(* PLC project 117_1_V0.5.project, CODESYS CODESYS V3.5 SP17 Patch 3 *)
(* stored: creationDateTime 1970-01-01T00:00:00, modificationDateTime 2026-03-26T18:14:32.4070562 *)

FUNCTION_BLOCK TimeManager
  VAR
    hTask : CmpIecTask.RTS_IEC_HANDLE;  (* Дескриптор (handle) задачи * ) *)
    result : CmpIecTask.RTS_IEC_RESULT;  (* Результат выполнения функций * ) *)
    pCurrentTaskInfo : POINTER TO CmpIecTask.Task_Info2;  (* Указатель на структуру с информацией о задаче * ) *)
    CurrentTaskInfo : CmpIecTask.Task_Info2;  (* Сама структура с данными * ) *)
    DateAndTime : DTU.GetDateAndTime;
    _dateAndTime : DT;
  END_VAR

            
// 1. Получаем дескриптор текущей задачи
hTask := CmpIecTask.IecTaskGetCurrent(pResult := ADR(result));

// 2. Если дескриптор получен успешно, запрашиваем информацию о задаче
IF hTask <> 0 THEN
    // IecTaskGetInfo3 возвращает указатель на структуру данных о задаче
    pCurrentTaskInfo := CmpIecTask.IecTaskGetInfo3(hIecTask := hTask, pResult := ADR(result));
    
    // 3. Если указатель действителен, копируем данные в нашу локальную переменную
    IF pCurrentTaskInfo <> 0 THEN
        CurrentTaskInfo := pCurrentTaskInfo^;
    END_IF 
END_IF


DateAndTime(xExecute := TRUE);
	IF DateAndTime.xDone THEN
		_dateAndTime := DateAndTime.dtDateAndTime;
		DateAndTime(xExecute := FALSE);
	END_IF

          

METHOD get_interval_time_type_UINT : UINT
  VAR_INPUT
    measurementUnits : MEASUREMENT_UNITS;
  END_VAR
                  CASE measurementUnits OF
	MS:                               
		get_interval_time_type_UINT  := DWORD_TO_UINT(CurrentTaskInfo.dwInterval / 1000);
	US:                                          
		get_interval_time_type_UINT  := DWORD_TO_uint(CurrentTaskInfo.dwInterval);
END_CASE


                
END_METHOD
END_FUNCTION_BLOCK
